PROGRAM maint_mode
VAR
	maint_mode: BOOL;
	
	u_3112_b_hmi_start_request: BOOL;
	u_3112_b_maint_request: BOOL;
	u_3112_b_hmi_speed_request: REAL;
	u_3112_b_maint_speed_request: REAL;
	u_3112_b_hmi_stop_request: BOOL;
	
	u_3212_b_hmi_start_request: BOOL;
	u_3212_b_maint_request: BOOL;
	u_3212_b_hmi_speed_request: REAL;
	u_3212_b_maint_speed_request: REAL;
	u_3212_b_hmi_stop_request: BOOL;

	u_3312_b_hmi_start_request: BOOL;
	u_3312_b_maint_request: BOOL;
	u_3312_b_hmi_speed_request: REAL;
	u_3312_b_maint_speed_request: REAL;
	u_3312_b_hmi_stop_request: BOOL;
	
	u_3405_b_hmi_start_request: BOOL;
	u_3405_b_maint_request: BOOL;
	u_3405_b_hmi_speed_request: REAL;
	u_3405_b_maint_speed_request: REAL;
	u_3405_b_hmi_stop_request: BOOL;
	
	u_3160_b_hmi_start_request: BOOL;
	u_3160_b_maint_request: BOOL;
	u_3160_b_hmi_speed_request: REAL;
	u_3160_b_maint_speed_request: REAL;
	u_3160_b_hmi_stop_request: BOOL;
	
	u_3260_b_hmi_start_request: BOOL;
	u_3260_b_maint_request: BOOL;
	u_3260_b_hmi_speed_request: REAL;
	u_3260_b_maint_speed_request: REAL;
	u_3260_b_hmi_stop_request: BOOL;
	
	u_3360_b_hmi_start_request: BOOL;
	u_3360_b_maint_request: BOOL;
	u_3360_b_hmi_speed_request: REAL;
	u_3360_b_maint_speed_request: REAL;
	u_3360_b_hmi_stop_request: BOOL;
	
	nv_3110_b_hmi_open_request: BOOL;
	nv_3110_b_hmi_close_request: BOOL;
	nv_3110_b_maint_request: BOOL;
	
	nv_3210_b_hmi_open_request: BOOL;
	nv_3210_b_hmi_close_request: BOOL;
	nv_3210_b_maint_request: BOOL;
	
	nv_3310_b_hmi_open_request: BOOL;
	nv_3310_b_hmi_close_request: BOOL;
	nv_3310_b_maint_request: BOOL;
	
	nv_3135_b_hmi_open_request: BOOL;
	nv_3135_b_hmi_close_request: BOOL;
	nv_3135_b_maint_request: BOOL;
	
	nv_3235_b_hmi_open_request: BOOL;
	nv_3235_b_hmi_close_request: BOOL;
	nv_3235_b_maint_request: BOOL;
	
	nv_3335_b_hmi_open_request: BOOL;
	nv_3335_b_hmi_close_request: BOOL;
	nv_3335_b_maint_request: BOOL;
	
	nv_3372_b_hmi_open_request: BOOL;
	nv_3372_b_hmi_close_request: BOOL;
	nv_3372_b_maint_request: BOOL;
	u_3370_b_hmi_start_request: BOOL;
	u_3370_b_maint_request: BOOL;
	u_3370_b_hmi_stop_request: BOOL;
	u_3370_b_hmi_speed_request: REAL;
	u_3370_b_maint_speed_request: REAL;
	nv_3162_b_hmi_open_request: BOOL;
	nv_3162_b_maint_request: BOOL;
	nv_3162_b_hmi_close_request: BOOL;
END_VAR

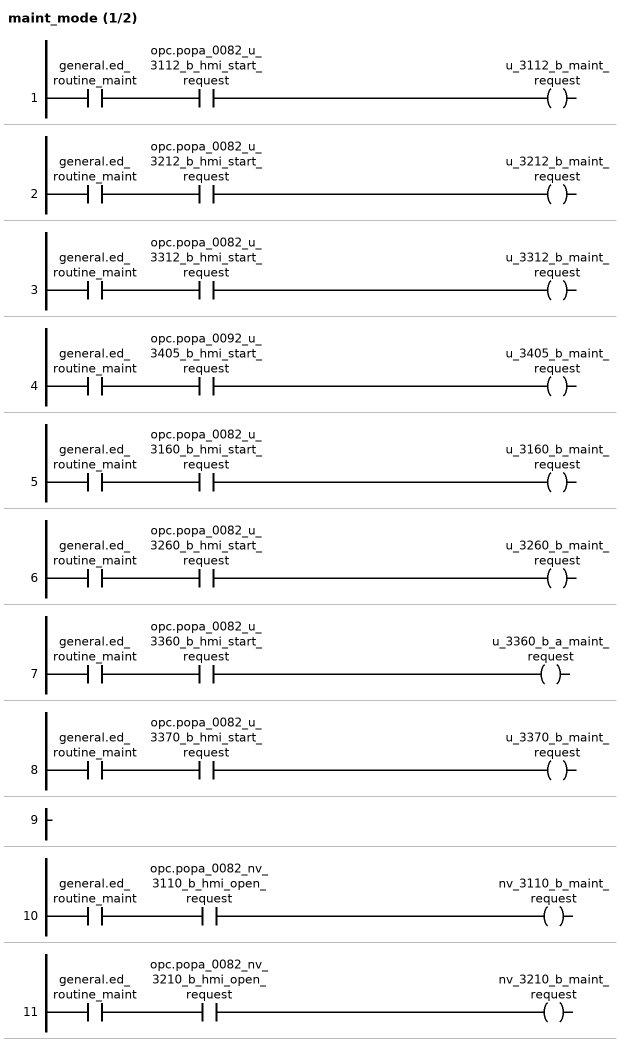
// NETWORK 1
u_3112_b_maint_request := general.ed_routine_maint AND opc.popa_0082_u_3112_b_hmi_start_request;

// NETWORK 2
u_3212_b_maint_request := general.ed_routine_maint AND opc.popa_0082_u_3212_b_hmi_start_request;

// NETWORK 3
u_3312_b_maint_request := general.ed_routine_maint AND opc.popa_0082_u_3312_b_hmi_start_request;

// NETWORK 4
u_3405_b_maint_request := general.ed_routine_maint AND opc.popa_0092_u_3405_b_hmi_start_request;

// NETWORK 5
u_3160_b_maint_request := general.ed_routine_maint AND opc.popa_0082_u_3160_b_hmi_start_request;

// NETWORK 6
u_3260_b_maint_request := general.ed_routine_maint AND opc.popa_0082_u_3260_b_hmi_start_request;

// NETWORK 7
u_3360_b_a_maint_request := general.ed_routine_maint AND opc.popa_0082_u_3360_b_hmi_start_request;

// NETWORK 8
u_3370_b_maint_request := general.ed_routine_maint AND opc.popa_0082_u_3370_b_hmi_start_request;

// NETWORK 9

// NETWORK 10
nv_3110_b_maint_request := general.ed_routine_maint AND opc.popa_0082_nv_3110_b_hmi_open_request;

// NETWORK 11
nv_3210_b_maint_request := general.ed_routine_maint AND opc.popa_0082_nv_3210_b_hmi_open_request;

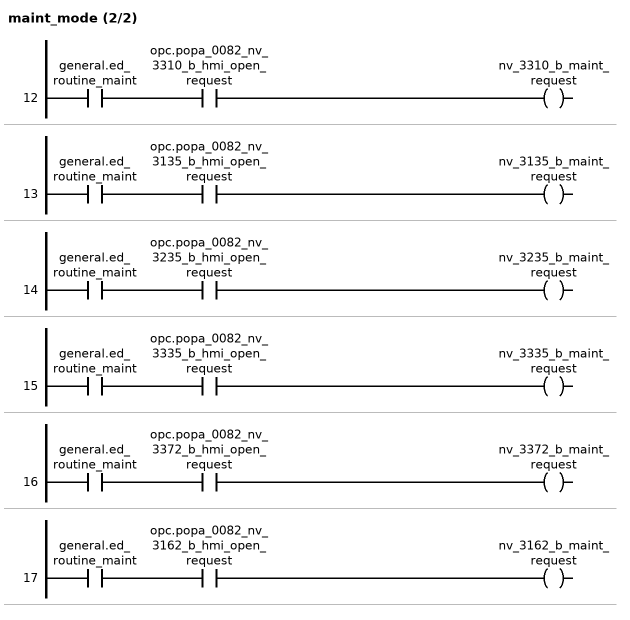
// NETWORK 12
nv_3310_b_maint_request := general.ed_routine_maint AND opc.popa_0082_nv_3310_b_hmi_open_request;

// NETWORK 13
nv_3135_b_maint_request := general.ed_routine_maint AND opc.popa_0082_nv_3135_b_hmi_open_request;

// NETWORK 14
nv_3235_b_maint_request := general.ed_routine_maint AND opc.popa_0082_nv_3235_b_hmi_open_request;

// NETWORK 15
nv_3335_b_maint_request := general.ed_routine_maint AND opc.popa_0082_nv_3335_b_hmi_open_request;

// NETWORK 16
nv_3372_b_maint_request := general.ed_routine_maint AND opc.popa_0082_nv_3372_b_hmi_open_request;

// NETWORK 17
nv_3162_b_maint_request := general.ed_routine_maint AND opc.popa_0082_nv_3162_b_hmi_open_request;

END_PROGRAM

(* stored: Version 1.1.0.1, ProductVersion 3.1.4024.15
   POU maint_mode: Id {fe91578f-e7b9-4e8e-a60b-a630302703f0}, SpecialFunc None *)
